(* CODESYS project Lift Structured Text New.project

Project tree, tasks and I/O mapping:
  CageTest : CODESYS Control Win V3, 3S - Smart Software Solutions GmbH, version 3.5.14.0
    application Application
      task CageTestTask (cyclic, interval t#20ms, priority 1) calls Simulatie, CageTestProgram
      visualisation Visualization
  DoorTest : CODESYS Control Win V3, 3S - Smart Software Solutions GmbH, version 3.5.14.0
    application Application
      libraries: Standard, * (System)
      task DoorTestTask (cyclic, interval t#20ms, priority 1) calls DoorTestProgram, Simulatie
      visualisation Visualization
  Elevator : CODESYS Control Win V3, 3S - Smart Software Solutions GmbH, version 3.5.14.0
    application Application
      libraries: Standard, * (System)
      task ElevatorTask (cyclic, interval t#20ms, priority 1) calls MainProgram, Simulatie
      visualisation Visualization
  Lift Besturing/
    program DoorTestProgram [ST]
    function block Door [ST]: goOpen, goClose, isClosed, cycle, initialaize, isOpen
    data type DoorStates
    program MainProgram [ST]
    function block Elevator [ST]: initialiaze, cycle
    data type CageStates
    function block Cage [ST]: initialaize, cycle, startTraveling, isUp, isDown, isTraveling
    program CageTestProgram [ST]
    data type ElevatorStates
  global variables GVL
  image pool ImagePool
  5ce3da45-db07-42e7-a21c-a00fff4ed8f6|C:\Users\Gerard\Desktop\MensenInLift.PNG
  5ce3da45-db07-42e7-a21c-a00fff4ed8f6|C:\Users\Gerard\Desktop\LiftDeur.PNG
  5ce3da45-db07-42e7-a21c-a00fff4ed8f6|C:\Users\Gerard\Desktop\Liftaandrijving.PNG
  5ce3da45-db07-42e7-a21c-a00fff4ed8f6|C:\Users\Gerard\Desktop\LiftDeurAandrijving.PNG
  Lift Simualtie/
    program Simulatie [ST]
  text list GlobalTextList
  visualisation Visualization
*)

// Lift Besturing/DoorStates
// Authour : G A Harkema
// Date:  february 15, 2017
// Version : 1.0
// States of the door
TYPE DoorStates :
(
	idle := 0,close, toOpen, open, toClose
);
END_TYPE

// Lift Besturing/CageStates
// Authour : G A Harkema
// Date:  february 15, 2017
// Version : 1.0
// States of the cage
TYPE CageStates :
(
	idle := 0, stationary, goUp, goDown  
);
END_TYPE

// Lift Besturing/ElevatorStates
// Authour : G A Harkema
// Date:  february 15, 2017
// Version : 1.0
// States of the cage
TYPE ElevatorStates :
(
	idle := 0, waitForChoise, closingDoor, traveling, openingDoor
);
END_TYPE

// GVL
VAR_GLOBAL
	Ix_BovenOproepKooi					: BOOL;
	Ix_BenedenOproepKooi				: BOOL;
	Ix_KooiGaNaarBoven					: BOOL;
	Ix_KooiGaNaarBeneden				: BOOL;
	Ix_KooiBoven						: BOOL;
	Ix_KooiBeneden						: BOOL;
	Qx_AandrijvingOmhoog				: BOOL;
	Qx_AandrijvingOmlaag				: BOOL;
	
	
	Ix_BenedenDeurOpen					: BOOL;
	Ix_BenedenDeurGesloten				: BOOL;
	Qx_BenedenDeurAandrijvingOpen		: BOOL;
	Qx_BenedenDeurAandrijvingSluiten	: BOOL;
	
	Ix_BovenDeurOpen					: BOOL;
	Ix_BovenDeurGesloten				: BOOL;
	Qx_BovenDeurAandrijvingOpen			: BOOL;
	Qx_BovenDeurAandrijvingSluiten		: BOOL;
	
	Ix_TestButton1						: BOOL;
	Ix_TestButton2						: BOOL;
	
	Qx_TestIndicator1					: BOOL;
	Qx_TestIndicator2					: BOOL;
	
END_VAR

// Lift Simualtie/Simulatie
// Programma		: Simulatie
// Project			: Lift
// Doel				: Simulatie functies voor de lift
// Auteur			: Gerard Harkema
// Versie			: 1.0
// Datum			: 15 oktober 2015

PROGRAM Simulatie
VAR

	Mw_PositieLiftInv					: INT := 0;
	Mw_PositieLift						: INT := 0;
	Mw_LiftBenedenCountValue			: INT := 250;

	Mw_BenedenPositieDeur				: INT := 0;
	Mw_BenedenPositieDeurCountValue		: INT := 100;

	Mw_BovenPositieDeur					: INT := 0;
	Mw_BovenPositieDeurCountValue		: INT := 100;

END_VAR


// Reizen lift omhoog
IF(GVL.Qx_AandrijvingOmhoog AND (NOT GVL.Ix_KooiBoven)) THEN
	Mw_PositieLiftInv := Mw_PositieLiftInv + 1;
END_IF

// Reizen lift omlaag
IF(GVL.Qx_AandrijvingOmlaag AND (NOT GVL.Ix_KooiBeneden)) THEN
	Mw_PositieLiftInv := Mw_PositieLiftInv - 1;
END_IF

Mw_PositieLift := Mw_LiftBenedenCountValue - Mw_PositieLiftInv;

// Detectie lift is boven
IF (Mw_PositieLiftInv >= Mw_LiftBenedenCountValue) THEN
	GVL.Ix_KooiBoven := TRUE;
ELSE
	GVL.Ix_KooiBoven := FALSE;	
END_IF
  

// Detectie lift is beneden
IF(Mw_PositieLiftInv <= 0) THEN
	GVL.Ix_KooiBeneden := TRUE;
ELSE
	GVL.Ix_KooiBeneden := FALSE;	
END_IF

// Inactief maken oproepknoppen
IF GVL.Ix_KooiBoven THEN
 Ix_BovenOproepKooi := FALSE;
 Ix_KooiGaNaarBoven := FALSE;
END_IF

IF GVL.Ix_KooiBeneden THEN
 Ix_BenedenOproepKooi := FALSE;
 Ix_KooiGaNaarBeneden := FALSE;
END_IF


//*********************************************
//                 Bovendeur
//*********************************************

// Bovendeur openen
IF(GVL.Qx_BovenDeurAandrijvingOpen AND (NOT GVL.Ix_BovenDeurOpen)) THEN
	Mw_BovenPositieDeur := Mw_BovenPositieDeur + 1;
END_IF

// Bovendeur sluiten
IF(GVL.Qx_BovenDeurAandrijvingSluiten AND (NOT GVL.Ix_BovenDeurGesloten)) THEN
	Mw_BovenPositieDeur := Mw_BovenPositieDeur - 1;
END_IF

IF (Mw_BovenPositieDeur >= Mw_BovenPositieDeurCountValue) THEN
	GVL.Ix_BovenDeurOpen := TRUE;
ELSE
	GVL.Ix_BovenDeurOpen := FALSE;	
END_IF
  

// Detectie bovendeur is gesloten
IF(Mw_BovenPositieDeur <= 0) THEN
	GVL.Ix_BovenDeurGesloten := TRUE;
ELSE
	GVL.Ix_BovenDeurGesloten := FALSE;	
END_IF

//*********************************************
//                 Benedendeur
//*********************************************

// Benedendeur openen
IF(GVL.Qx_BenedenDeurAandrijvingOpen AND (NOT GVL.Ix_BenedenDeurOpen)) THEN
	Mw_BenedenPositieDeur := Mw_BenedenPositieDeur + 1;
END_IF

// Benedendeur sluiten
IF(GVL.Qx_BenedenDeurAandrijvingSluiten AND (NOT GVL.Ix_BenedenDeurGesloten)) THEN
	Mw_BenedenPositieDeur := Mw_BenedenPositieDeur - 1;
END_IF

// Detectie Benedendeur is open
IF (Mw_BenedenPositieDeur >= Mw_BenedenPositieDeurCountValue) THEN
	GVL.Ix_BenedenDeurOpen := TRUE;
ELSE
	GVL.Ix_BenedenDeurOpen := FALSE;	
END_IF

// Detectie Benedendeur is gesloten
IF(Mw_BenedenPositieDeur <= 0) THEN
	GVL.Ix_BenedenDeurGesloten := TRUE;
ELSE
	GVL.Ix_BenedenDeurGesloten := FALSE;	
END_IF

END_PROGRAM

// Lift Besturing/CageTestProgram
// Authour : G A Harkema
// Date:  february 15, 2017
// Version : 1.0
// Testprogram for the cage

PROGRAM CageTestProgram
VAR
	theCage				: Cage;
	firstRun		 	: BOOL := TRUE;
END_VAR

IF firstRun THEN
	// make references to I/O
	theCage.initialaize();
	firstRun := FALSE;
END_IF

// Update inputs of the objects
theCage.xCageIsUp := gvl.Ix_KooiBoven;
theCage.xCageIsDown := gvl.Ix_KooiBeneden;

theCage.cycle();

// Update Outputs from the object
gvl.Qx_AandrijvingOmhoog := TheCage.xTransmissionUp;
gvl.Qx_AandrijvingOmlaag := TheCage.xTransmissionDown;

Qx_TestIndicator1 := theCage.isTraveling();

IF NOT theCage.isTraveling() THEN
	IF Ix_TestButton1 THEN // Handle button event
		Ix_TestButton1 := FALSE;
		theCage.startTraveling();
	END_IF
END_IF

END_PROGRAM

// Lift Besturing/Cage
// Authour : G A Harkema
// Date:  february 15, 2017
// Version : 1.0
// Class of the elevator

FUNCTION_BLOCK Cage
VAR
	eState								: CageStates := CageStates.idle;
END_VAR

VAR_INPUT
	xCageIsUp							: BOOL; 
	xCageIsDown							: BOOL; 
END_VAR

VAR_OUTPUT
	xTransmissionUp						: BOOL; 
	xTransmissionDown					: BOOL; 
END_VAR

// Statemachine of the cage
CASE eState OF

	CageStates.idle:
		xTransmissionDown := TRUE;  // powerup sequence
		eState := CageStates.goDown;


	CageStates.goDown:
		IF xCageIsDown THEN  // Handle downstair event
			xTransmissionDown := FALSE;
			eState := CageStates.stationary;
		END_IF
	
	CageStates.goUp:
		IF xCageIsUp THEN  // Handle upstairs event
			xTransmissionUp := FALSE;
			eState := CageStates.stationary;
		END_IF

	
END_CASE

// initialaize I/O
METHOD initialaize
VAR_INPUT
END_VAR
// Set default values
xTransmissionUp 	:= FALSE;
xTransmissionDown 	:= FALSE;
END_METHOD

// Update statemachine and I/O
METHOD cycle
VAR_INPUT
END_VAR
THIS^();
END_METHOD

// start traveling of cage
METHOD startTraveling
VAR_INPUT
END_VAR
IF eState = CageStates.stationary THEN
	
	// Check position of the cage and handle
	IF isUp() THEN
		xTransmissionDown := TRUE;
		eState := CageStates.goDown;
	END_IF
	
	IF isDown() THEN
		xTransmissionUp := TRUE;
		eState := CageStates.goUp;
	END_IF
	
END_IF
END_METHOD

// check upstairs methode
METHOD PUBLIC isUp : BOOL
VAR_INPUT
END_VAR
isUp := xCageIsUp;
END_METHOD

// check downstairs methode
METHOD PUBLIC isDown : BOOL
VAR_INPUT
END_VAR
isDown := xCageIsDown;
END_METHOD

// check traveling methode
METHOD PUBLIC isTraveling : BOOL
VAR_INPUT
END_VAR
isTraveling := NOT(eState = CageStates.stationary);
END_METHOD

END_FUNCTION_BLOCK

// Lift Besturing/Elevator
// Authour : G A Harkema
// Date:  february 15, 2017
// Version : 1.0
// Class of the elevator

FUNCTION_BLOCK Elevator
VAR_INPUT
	doorUpstairs   		: Door;
	doorDownstairs   	: Door;
	theCage				: Cage;
	initialiazed	 	: BOOL := FALSE;
	eState				: ElevatorStates := ElevatorStates.idle;
END_VAR

IF initialiazed THEN
	// Update statemachines and I/O
	doorUpstairs.cycle();
	doorDownstairs.cycle();
	theCage.cycle();
END_IF

METHOD initialiaze
VAR_INPUT
END_VAR
// make references to I/O
theCage.initialaize();
doorUpstairs.initialaize();
doorDownstairs.initialaize();

initialiazed := TRUE;
END_METHOD

// Update statemachine and I/O
METHOD cycle
VAR_INPUT
END_VAR
THIS^();

// Update inputs of the objects
theCage.xCageIsUp := gvl.Ix_KooiBoven;
theCage.xCageIsDown := gvl.Ix_KooiBeneden;

doorDownstairs.xDoorIsOpen := gvl.Ix_BenedenDeurOpen;
doorDownstairs.xDoorIsClose := gvl.Ix_BenedenDeurGesloten;

doorUpstairs.xDoorIsOpen := gvl.Ix_BovenDeurOpen;
doorUpstairs.xDoorIsClose := gvl.Ix_BovenDeurGesloten;

	
// Handle state machine
CASE eState OF
	ElevatorStates.idle:
		eState := ElevatorStates.waitForChoise;

	ElevatorStates.waitForChoise:
		IF theCage.isUp() THEN  // handle choise
			IF Ix_KooiGaNaarBeneden OR Ix_BenedenOproepKooi THEN
				doorUpstairs.goClose();
				eState := ElevatorStates.closingDoor;
			END_IF
		END_IF
		
		IF theCage.isDown() THEN
			IF Ix_KooiGaNaarBoven OR Ix_BovenOproepKooi THEN
				doorDownstairs.goClose();
				eState := ElevatorStates.closingDoor;
			END_IF
		END_IF

	ElevatorStates.closingDoor:
		IF doorUpstairs.isClosed() AND doorDownstairs.isClosed() THEN // handle doors closed
			theCage.startTraveling();
			eState := ElevatorStates.traveling;
		END_IF
	
	ElevatorStates.traveling:
		IF NOT theCage.isTraveling() THEN // handle arriving of cage
			IF theCage.isUp()  THEN
				doorUpstairs.goOpen();
				eState := ElevatorStates.openingDoor;
			END_IF
	
			IF theCage.isDown() THEN
				doorDownstairs.goOpen();
				eState := ElevatorStates.openingDoor;
			END_IF
		END_IF;

	ElevatorStates.openingDoor:
		IF doorUpstairs.isOpen() OR doorDownstairs.isOpen() THEN // Handle door open
			eState := ElevatorStates.waitForChoise;
		END_IF
END_CASE

// Update Outputs from the object
gvl.Qx_AandrijvingOmhoog := TheCage.xTransmissionUp;
gvl.Qx_AandrijvingOmlaag := TheCage.xTransmissionDown;

gvl.Qx_BenedenDeurAandrijvingOpen := doorDownstairs.xDoorOpening;
gvl.Qx_BenedenDeurAandrijvingSluiten := doorDownstairs.xDoorClosing;

gvl.Qx_BovenDeurAandrijvingOpen := doorUpstairs.xDoorOpening;
gvl.Qx_BovenDeurAandrijvingSluiten := doorUpstairs.xDoorClosing;
END_METHOD

END_FUNCTION_BLOCK

// Lift Besturing/Door
// Authour : G A Harkema
// Date:  february 15, 2017
// Version : 1.0
// Class of the door

FUNCTION_BLOCK Door
VAR
	eState							: DoorStates := DoorStates.idle;
END_VAR

VAR_INPUT
	xDoorIsOpen						: BOOL; 
	xDoorIsClose					: BOOL; 
END_VAR

VAR_OUTPUT
	xDoorOpening					: BOOL; 
	xDoorClosing					: BOOL; 
END_VAR

// Statemachine of the door
CASE eState OF
	DoorStates.toOpen :
		IF xDoorIsOpen THEN  // handle open event
			xDoorOpening := FALSE;
			eState := DoorStates.open;
		END_IF
	
	DoorStates.toClose :
		IF xDoorIsClose THEN // handle close event
			xDoorClosing := FALSE;
			eState := DoorStates.close;
		END_IF
	
END_CASE

// start door open action methode
METHOD PUBLIC goOpen
VAR_INPUT
END_VAR
// Trigger door
IF eState = DoorStates.close THEN
	eState := DoorStates.toOpen;  // Hnadle event
	xDoorOpening := TRUE;
END_IF
END_METHOD

// start close door action method
METHOD PUBLIC goClose
VAR_INPUT
END_VAR
// Trigger door when open
IF eState = DoorStates.open THEN
	eState := DoorStates.toClose;  // Handle event
	xDoorClosing := TRUE;
END_IF


// Trigger door when close
IF eState = DoorStates.idle THEN
	eState := DoorStates.toClose; // Hnadle event
	xDoorClosing := TRUE;
END_IF
END_METHOD

// check door closed method
METHOD PUBLIC isClosed : BOOL
VAR_INPUT
END_VAR
isClosed := eState = DoorStates.close;
END_METHOD

// Update statemachine and I/O
METHOD cycle
VAR_INPUT
END_VAR
THIS^();
END_METHOD

// initialaize I/O
METHOD initialaize
VAR_INPUT
END_VAR

xDoorOpening := FALSE;
xDoorClosing := FALSE;
	

// Close the door	
goClose();
END_METHOD

// check door opened method
METHOD isOpen : BOOL
VAR_INPUT
END_VAR
isOpen := eState = DoorStates.open;
END_METHOD

END_FUNCTION_BLOCK

// Lift Besturing/DoorTestProgram
// Authour : G A Harkema
// Date:  february 15, 2017
// Version : 1.0
// Testprogram for the doors

PROGRAM DoorTestProgram
VAR
	doorUpstairs   		: Door;
	doorDownstairs   	: Door;
	firstRun		 	: BOOL := TRUE;
END_VAR

IF firstRun THEN
	// make references to I/O
	doorUpstairs.initialaize();
	doorDownstairs.initialaize();
	firstRun := FALSE;
END_IF

// Update inputs of the objects
doorDownstairs.xDoorIsOpen := gvl.Ix_BenedenDeurOpen;
doorDownstairs.xDoorIsClose := gvl.Ix_BenedenDeurGesloten;

doorUpstairs.xDoorIsOpen := gvl.Ix_BovenDeurOpen;
doorUpstairs.xDoorIsClose := gvl.Ix_BovenDeurGesloten;

// update I/O
doorUpstairs.cycle();
doorDownstairs.cycle();

// Update Outputs from the object
gvl.Qx_BenedenDeurAandrijvingOpen := doorDownstairs.xDoorOpening;
gvl.Qx_BenedenDeurAandrijvingSluiten := doorDownstairs.xDoorClosing;

gvl.Qx_BovenDeurAandrijvingOpen := doorUpstairs.xDoorOpening;
gvl.Qx_BovenDeurAandrijvingSluiten := doorUpstairs.xDoorClosing;

IF Ix_TestButton1 THEN
	Ix_TestButton1 := FALSE; // Handle button event
	doorUpstairs.goOpen();
	doorDownstairs.goClose();
END_IF

IF Ix_TestButton2 THEN
	Ix_TestButton2 := FALSE; // Handle button event
	doorUpstairs.goClose();
	doorDownstairs.goOpen();
END_IF

END_PROGRAM

// Lift Besturing/MainProgram
// Authour : G A Harkema
// Date:  february 15, 2017
// Version : 1.0
// Main program of the elevator

PROGRAM MainProgram
VAR
	// only one object is created in the main program
	theElevator			: Elevator;
	firstRun		 	: BOOL := TRUE;
END_VAR

IF firstRun THEN
	theElevator.initialiaze ();
	firstRun := FALSE;
END_IF


// update statemachines and I/O
theElevator.cycle();

END_PROGRAM

// CageTest/Application/Visualization
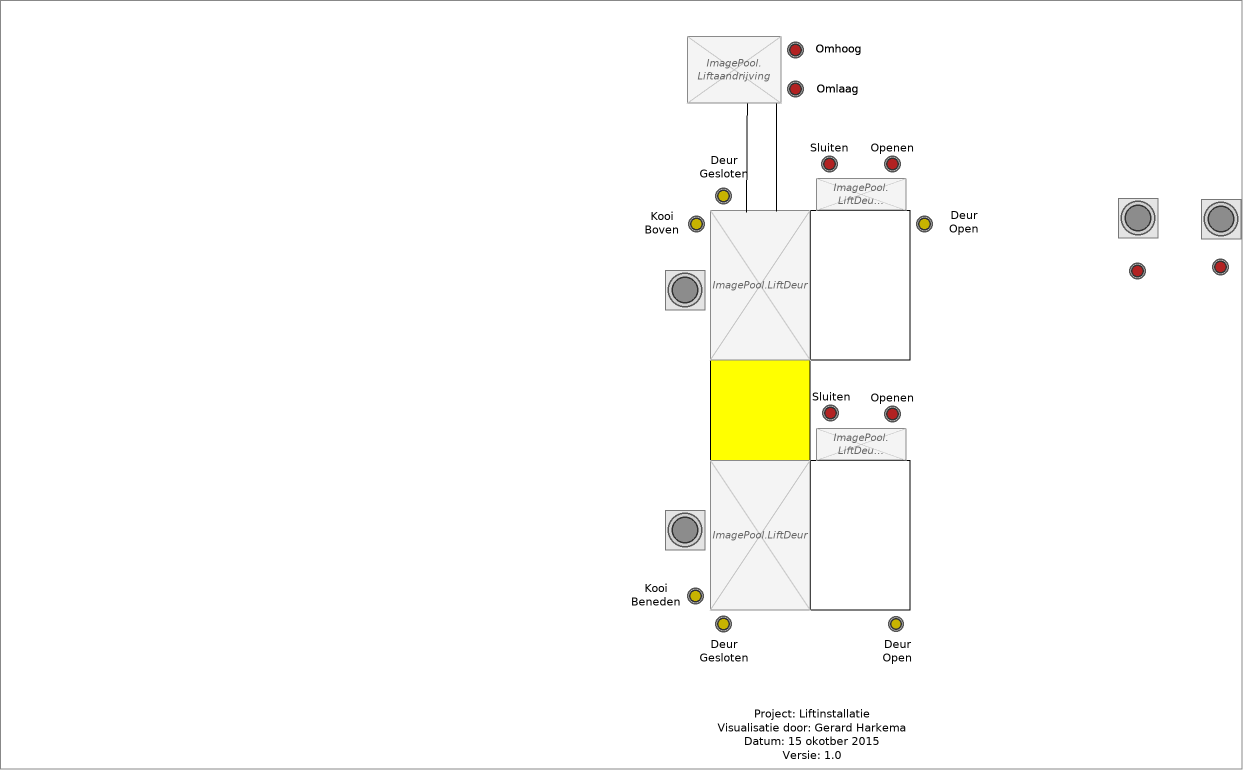
VISUALIZATION Visualization  // 1243x770
    Rectangle (810,460 100x150)
    Rectangle (810,210 100x150)
    Rectangle (710,210 100x400)
    PushSwitch (665,270 40x40), tooltip "Oproep Boven", variable: Ix_BovenOproepKooi, behaviour: TOGGLE, style: Switch-PushSwitch-Gray
    PushSwitch (665,510 40x40), tooltip "Oproep Beneden", variable: Ix_BenedenOproepKooi, behaviour: TOGGLE, style: Switch-PushSwitch-Gray
    Group (710,210 100x150)
        p2738717112: Simulatie.Mw_PositieLift
        Rectangle (0,0 100x150)
        Image (6,0 89x150), image: ImagePool.MensenInLift
        PushSwitch (5,100 30x30), tooltip "Ga naar beneden", variable: Ix_KooiGaNaarBeneden, behaviour: TOGGLE, style: Switch-PushSwitch-Gray
        PushSwitch (5,60 30x30), tooltip "Ga naar Boven", variable: Ix_KooiGaNaarBoven, behaviour: TOGGLE, style: Switch-PushSwitch-Gray
    Rectangle (710,210 100x150)
    Image (716,210 89x150), image: ImagePool.MensenInLift
    PushSwitch (715,310 30x30), tooltip "Ga naar beneden", variable: Ix_KooiGaNaarBeneden, behaviour: TOGGLE, style: Switch-PushSwitch-Gray
    PushSwitch (715,270 30x30), tooltip "Ga naar Boven", variable: Ix_KooiGaNaarBoven, behaviour: TOGGLE, style: Switch-PushSwitch-Gray
    Lamp1 (714,186 19x20), variable: Ix_BovenDeurGesloten, style: Lamp-Lamp1-Yellow
    Lamp1 (915,214 19x20), variable: Ix_BovenDeurOpen, style: Lamp-Lamp1-Yellow
    Lamp1 (687,214 19x20), variable: Ix_KooiBoven, style: Lamp-Lamp1-Yellow
    Lamp1 (686,586 19x20), variable: Ix_KooiBeneden, style: Lamp-Lamp1-Yellow
    Lamp1 (714,614 19x20), variable: Ix_BenedenDeurGesloten, style: Lamp-Lamp1-Yellow
    Lamp1 (887,614 18x20), variable: Ix_BenedenDeurOpen, style: Lamp-Lamp1-Yellow
    Label (682,152 84x30), "Deur Gesloten"
    Label (937,207 54x30), "Deur Open"
    Label (640,208 44x30), "Kooi Boven"
    Label (629,580 54x30), "Kooi Beneden"
    Label (693,636 62x30), "Deur Gesloten"
    Label (875,636 45x30), "Deur Open"
    Group (710,210 100x150)
        p3560616238: Simulatie.Mw_BovenPositieDeur
        Rectangle (0,0 100x150)
        Image (0,0 100x150), image: ImagePool.LiftDeur
    Group (710,460 100x150)
        p3560616238: Simulatie.Mw_BenedenPositieDeur
        Rectangle (0,0 100x150)
        Image (0,0 100x150), image: ImagePool.LiftDeur
    Line (747,83) (746,212)
    Line (776,82) (776,211)
    Group (687,34 182x70)
        Image (0,2 94x67), image: ImagePool.Liftaandrijving
        Lamp1 (99,6 19x20), variable: Qx_AandrijvingOmhoog, style: Lamp-Lamp1-Red
        Lamp1 (99,45 19x20), variable: Qx_AandrijvingOmlaag, style: Lamp-Lamp1-Red
        Label (121,0 61x30), "Omhoog"
        Label (123,40 55x30), "Omlaag"
    Image (687,36 94x67), image: ImagePool.Liftaandrijving
    Lamp1 (786,40 19x20), variable: Qx_AandrijvingOmhoog, style: Lamp-Lamp1-Red
    Lamp1 (786,79 19x20), variable: Qx_AandrijvingOmlaag, style: Lamp-Lamp1-Red
    Label (808,34 61x30), "Omhoog"
    Label (810,74 55x30), "Omlaag"
    Group (816,154 90x56)
        Image (0,24 90x32), image: ImagePool.LiftDeurAandrijving
        Lamp1 (4,0 19x20), variable: Qx_BovenDeurAandrijvingSluiten, style: Lamp-Lamp1-Red
        Lamp1 (67,0 19x20), variable: Qx_BovenDeurAandrijvingOpen, style: Lamp-Lamp1-Red
    Image (816,178 90x32), image: ImagePool.LiftDeurAandrijving
    Lamp1 (820,154 19x20), variable: Qx_BovenDeurAandrijvingSluiten, style: Lamp-Lamp1-Red
    Lamp1 (883,154 19x20), variable: Qx_BovenDeurAandrijvingOpen, style: Lamp-Lamp1-Red
    Group (816,403 90x57)
        Image (0,25 90x32), image: ImagePool.LiftDeurAandrijving
        Lamp1 (5,0 19x20), variable: Qx_BenedenDeurAandrijvingSluiten, style: Lamp-Lamp1-Red
        Lamp1 (67,1 19x20), variable: Qx_BenedenDeurAandrijvingOpen, style: Lamp-Lamp1-Red
    Image (816,428 90x32), image: ImagePool.LiftDeurAandrijving
    Lamp1 (821,403 19x20), variable: Qx_BenedenDeurAandrijvingSluiten, style: Lamp-Lamp1-Red
    Lamp1 (883,404 19x20), variable: Qx_BenedenDeurAandrijvingOpen, style: Lamp-Lamp1-Red
    Label (812,382 39x30), "Sluiten"
    Label (810,133 39x30), "Sluiten"
    Label (867,383 51x30), "Openen"
    Label (867,133 51x30), "Openen"
    Label (712,701 200x67), "Project: Liftinstallatie Visualisatie door: Gerard Harkema Datum: 15 okotber 2015 Versie: 1.0"
    PushSwitch (1118,198 40x40), tooltip "Test Button 1", variable: Ix_TestButton1, behaviour: TOGGLE, style: Switch-PushSwitch-Gray
    PushSwitch (1201,199 40x40), tooltip "Test Button 2", variable: Ix_TestButton2, behaviour: TOGGLE, style: Switch-PushSwitch-Gray
    Lamp1 (1128,261 19x20), variable: Qx_TestIndicator1, style: Lamp-Lamp1-Red
    Lamp1 (1211,257 19x20), variable: Qx_TestIndicator2, style: Lamp-Lamp1-Red
END_VISUALIZATION

// DoorTest/Application/Visualization
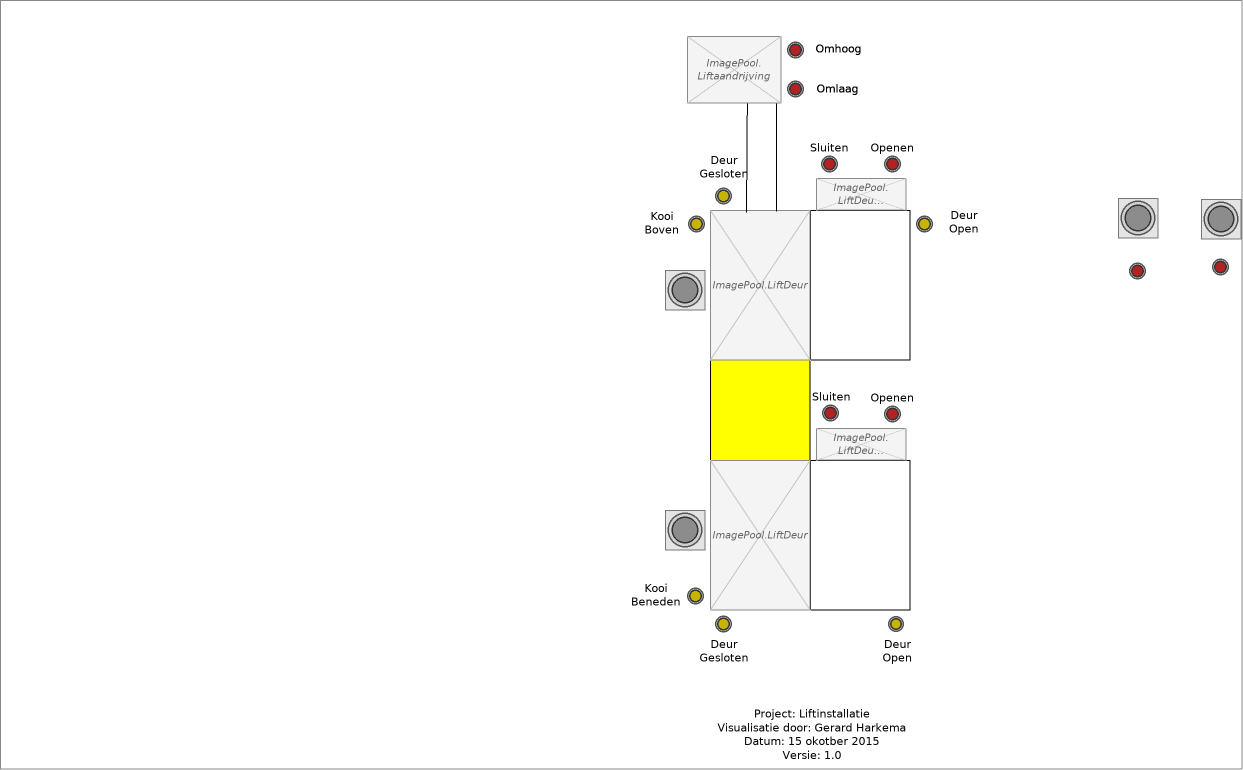
VISUALIZATION Visualization  // 1243x770
    Rectangle (810,460 100x150)
    Rectangle (810,210 100x150)
    Rectangle (710,210 100x400)
    PushSwitch (665,270 40x40), tooltip "Oproep Boven", variable: Ix_BovenOproepKooi, behaviour: TOGGLE, style: Switch-PushSwitch-Gray
    PushSwitch (665,510 40x40), tooltip "Oproep Beneden", variable: Ix_BenedenOproepKooi, behaviour: TOGGLE, style: Switch-PushSwitch-Gray
    Group (710,210 100x150)
        p2738717112: Simulatie.Mw_PositieLift
        Rectangle (0,0 100x150)
        Image (6,0 89x150), image: ImagePool.MensenInLift
        PushSwitch (5,100 30x30), tooltip "Ga naar beneden", variable: Ix_KooiGaNaarBeneden, behaviour: TOGGLE, style: Switch-PushSwitch-Gray
        PushSwitch (5,60 30x30), tooltip "Ga naar Boven", variable: Ix_KooiGaNaarBoven, behaviour: TOGGLE, style: Switch-PushSwitch-Gray
    Rectangle (710,210 100x150)
    Image (716,210 89x150), image: ImagePool.MensenInLift
    PushSwitch (715,310 30x30), tooltip "Ga naar beneden", variable: Ix_KooiGaNaarBeneden, behaviour: TOGGLE, style: Switch-PushSwitch-Gray
    PushSwitch (715,270 30x30), tooltip "Ga naar Boven", variable: Ix_KooiGaNaarBoven, behaviour: TOGGLE, style: Switch-PushSwitch-Gray
    Lamp1 (714,186 19x20), variable: Ix_BovenDeurGesloten, style: Lamp-Lamp1-Yellow
    Lamp1 (915,214 19x20), variable: Ix_BovenDeurOpen, style: Lamp-Lamp1-Yellow
    Lamp1 (687,214 19x20), variable: Ix_KooiBoven, style: Lamp-Lamp1-Yellow
    Lamp1 (686,586 19x20), variable: Ix_KooiBeneden, style: Lamp-Lamp1-Yellow
    Lamp1 (714,614 19x20), variable: Ix_BenedenDeurGesloten, style: Lamp-Lamp1-Yellow
    Lamp1 (887,614 18x20), variable: Ix_BenedenDeurOpen, style: Lamp-Lamp1-Yellow
    Label (682,152 84x30), "Deur Gesloten"
    Label (937,207 54x30), "Deur Open"
    Label (640,208 44x30), "Kooi Boven"
    Label (629,580 54x30), "Kooi Beneden"
    Label (693,636 62x30), "Deur Gesloten"
    Label (875,636 45x30), "Deur Open"
    Group (710,210 100x150)
        p3560616238: Simulatie.Mw_BovenPositieDeur
        Rectangle (0,0 100x150)
        Image (0,0 100x150), image: ImagePool.LiftDeur
    Group (710,460 100x150)
        p3560616238: Simulatie.Mw_BenedenPositieDeur
        Rectangle (0,0 100x150)
        Image (0,0 100x150), image: ImagePool.LiftDeur
    Line (747,83) (746,212)
    Line (776,82) (776,211)
    Group (687,34 182x70)
        Image (0,2 94x67), image: ImagePool.Liftaandrijving
        Lamp1 (99,6 19x20), variable: Qx_AandrijvingOmhoog, style: Lamp-Lamp1-Red
        Lamp1 (99,45 19x20), variable: Qx_AandrijvingOmlaag, style: Lamp-Lamp1-Red
        Label (121,0 61x30), "Omhoog"
        Label (123,40 55x30), "Omlaag"
    Image (687,36 94x67), image: ImagePool.Liftaandrijving
    Lamp1 (786,40 19x20), variable: Qx_AandrijvingOmhoog, style: Lamp-Lamp1-Red
    Lamp1 (786,79 19x20), variable: Qx_AandrijvingOmlaag, style: Lamp-Lamp1-Red
    Label (808,34 61x30), "Omhoog"
    Label (810,74 55x30), "Omlaag"
    Group (816,154 90x56)
        Image (0,24 90x32), image: ImagePool.LiftDeurAandrijving
        Lamp1 (4,0 19x20), variable: Qx_BovenDeurAandrijvingSluiten, style: Lamp-Lamp1-Red
        Lamp1 (67,0 19x20), variable: Qx_BovenDeurAandrijvingOpen, style: Lamp-Lamp1-Red
    Image (816,178 90x32), image: ImagePool.LiftDeurAandrijving
    Lamp1 (820,154 19x20), variable: Qx_BovenDeurAandrijvingSluiten, style: Lamp-Lamp1-Red
    Lamp1 (883,154 19x20), variable: Qx_BovenDeurAandrijvingOpen, style: Lamp-Lamp1-Red
    Group (816,403 90x57)
        Image (0,25 90x32), image: ImagePool.LiftDeurAandrijving
        Lamp1 (5,0 19x20), variable: Qx_BenedenDeurAandrijvingSluiten, style: Lamp-Lamp1-Red
        Lamp1 (67,1 19x20), variable: Qx_BenedenDeurAandrijvingOpen, style: Lamp-Lamp1-Red
    Image (816,428 90x32), image: ImagePool.LiftDeurAandrijving
    Lamp1 (821,403 19x20), variable: Qx_BenedenDeurAandrijvingSluiten, style: Lamp-Lamp1-Red
    Lamp1 (883,404 19x20), variable: Qx_BenedenDeurAandrijvingOpen, style: Lamp-Lamp1-Red
    Label (812,382 39x30), "Sluiten"
    Label (810,133 39x30), "Sluiten"
    Label (867,383 51x30), "Openen"
    Label (867,133 51x30), "Openen"
    Label (712,701 200x67), "Project: Liftinstallatie Visualisatie door: Gerard Harkema Datum: 15 okotber 2015 Versie: 1.0"
    PushSwitch (1118,198 40x40), tooltip "Test Button 1", variable: Ix_TestButton1, behaviour: TOGGLE, style: Switch-PushSwitch-Gray
    PushSwitch (1201,199 40x40), tooltip "Test Button 2", variable: Ix_TestButton2, behaviour: TOGGLE, style: Switch-PushSwitch-Gray
    Lamp1 (1128,261 19x20), variable: Qx_TestIndicator1, style: Lamp-Lamp1-Red
    Lamp1 (1211,257 19x20), variable: Qx_TestIndicator2, style: Lamp-Lamp1-Red
END_VISUALIZATION

// /Visualization
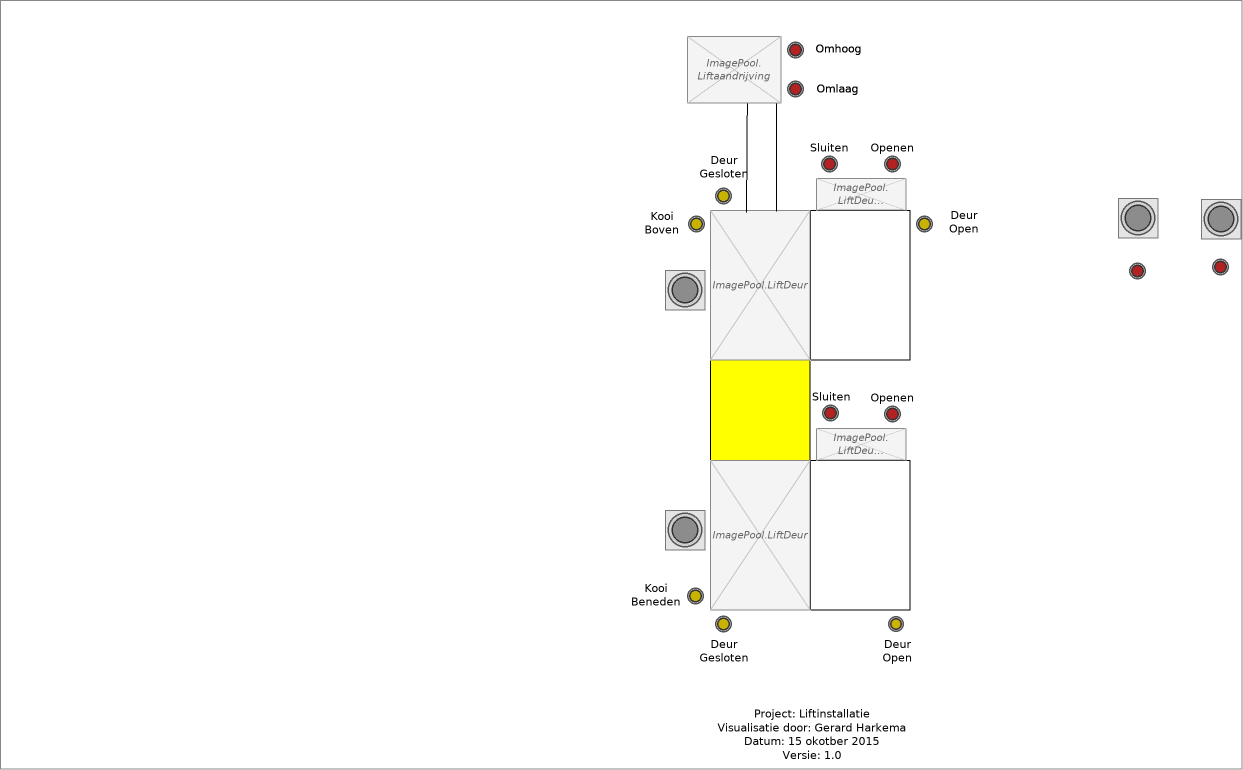
VISUALIZATION Visualization  // 1243x770
    Rectangle (810,460 100x150)
    Rectangle (810,210 100x150)
    Rectangle (710,210 100x400)
    PushSwitch (665,270 40x40), tooltip "Oproep Boven", variable: Ix_BovenOproepKooi, behaviour: TOGGLE, style: Switch-PushSwitch-Gray
    PushSwitch (665,510 40x40), tooltip "Oproep Beneden", variable: Ix_BenedenOproepKooi, behaviour: TOGGLE, style: Switch-PushSwitch-Gray
    Group (710,210 100x150)
        p2738717112: Simulatie.Mw_PositieLift
        Rectangle (0,0 100x150)
        Image (6,0 89x150), image: ImagePool.MensenInLift
        PushSwitch (5,100 30x30), tooltip "Ga naar beneden", variable: Ix_KooiGaNaarBeneden, behaviour: TOGGLE, style: Switch-PushSwitch-Gray
        PushSwitch (5,60 30x30), tooltip "Ga naar Boven", variable: Ix_KooiGaNaarBoven, behaviour: TOGGLE, style: Switch-PushSwitch-Gray
    Rectangle (710,210 100x150)
    Image (716,210 89x150), image: ImagePool.MensenInLift
    PushSwitch (715,310 30x30), tooltip "Ga naar beneden", variable: Ix_KooiGaNaarBeneden, behaviour: TOGGLE, style: Switch-PushSwitch-Gray
    PushSwitch (715,270 30x30), tooltip "Ga naar Boven", variable: Ix_KooiGaNaarBoven, behaviour: TOGGLE, style: Switch-PushSwitch-Gray
    Lamp1 (714,186 19x20), variable: Ix_BovenDeurGesloten, style: Lamp-Lamp1-Yellow
    Lamp1 (915,214 19x20), variable: Ix_BovenDeurOpen, style: Lamp-Lamp1-Yellow
    Lamp1 (687,214 19x20), variable: Ix_KooiBoven, style: Lamp-Lamp1-Yellow
    Lamp1 (686,586 19x20), variable: Ix_KooiBeneden, style: Lamp-Lamp1-Yellow
    Lamp1 (714,614 19x20), variable: Ix_BenedenDeurGesloten, style: Lamp-Lamp1-Yellow
    Lamp1 (887,614 18x20), variable: Ix_BenedenDeurOpen, style: Lamp-Lamp1-Yellow
    Label (682,152 84x30), "Deur Gesloten"
    Label (937,207 54x30), "Deur Open"
    Label (640,208 44x30), "Kooi Boven"
    Label (629,580 54x30), "Kooi Beneden"
    Label (693,636 62x30), "Deur Gesloten"
    Label (875,636 45x30), "Deur Open"
    Group (710,210 100x150)
        p3560616238: Simulatie.Mw_BovenPositieDeur
        Rectangle (0,0 100x150)
        Image (0,0 100x150), image: ImagePool.LiftDeur
    Group (710,460 100x150)
        p3560616238: Simulatie.Mw_BenedenPositieDeur
        Rectangle (0,0 100x150)
        Image (0,0 100x150), image: ImagePool.LiftDeur
    Line (747,83) (746,212)
    Line (776,82) (776,211)
    Group (687,34 182x70)
        Image (0,2 94x67), image: ImagePool.Liftaandrijving
        Lamp1 (99,6 19x20), variable: Qx_AandrijvingOmhoog, style: Lamp-Lamp1-Red
        Lamp1 (99,45 19x20), variable: Qx_AandrijvingOmlaag, style: Lamp-Lamp1-Red
        Label (121,0 61x30), "Omhoog"
        Label (123,40 55x30), "Omlaag"
    Image (687,36 94x67), image: ImagePool.Liftaandrijving
    Lamp1 (786,40 19x20), variable: Qx_AandrijvingOmhoog, style: Lamp-Lamp1-Red
    Lamp1 (786,79 19x20), variable: Qx_AandrijvingOmlaag, style: Lamp-Lamp1-Red
    Label (808,34 61x30), "Omhoog"
    Label (810,74 55x30), "Omlaag"
    Group (816,154 90x56)
        Image (0,24 90x32), image: ImagePool.LiftDeurAandrijving
        Lamp1 (4,0 19x20), variable: Qx_BovenDeurAandrijvingSluiten, style: Lamp-Lamp1-Red
        Lamp1 (67,0 19x20), variable: Qx_BovenDeurAandrijvingOpen, style: Lamp-Lamp1-Red
    Image (816,178 90x32), image: ImagePool.LiftDeurAandrijving
    Lamp1 (820,154 19x20), variable: Qx_BovenDeurAandrijvingSluiten, style: Lamp-Lamp1-Red
    Lamp1 (883,154 19x20), variable: Qx_BovenDeurAandrijvingOpen, style: Lamp-Lamp1-Red
    Group (816,403 90x57)
        Image (0,25 90x32), image: ImagePool.LiftDeurAandrijving
        Lamp1 (5,0 19x20), variable: Qx_BenedenDeurAandrijvingSluiten, style: Lamp-Lamp1-Red
        Lamp1 (67,1 19x20), variable: Qx_BenedenDeurAandrijvingOpen, style: Lamp-Lamp1-Red
    Image (816,428 90x32), image: ImagePool.LiftDeurAandrijving
    Lamp1 (821,403 19x20), variable: Qx_BenedenDeurAandrijvingSluiten, style: Lamp-Lamp1-Red
    Lamp1 (883,404 19x20), variable: Qx_BenedenDeurAandrijvingOpen, style: Lamp-Lamp1-Red
    Label (812,382 39x30), "Sluiten"
    Label (810,133 39x30), "Sluiten"
    Label (867,383 51x30), "Openen"
    Label (867,133 51x30), "Openen"
    Label (712,701 200x67), "Project: Liftinstallatie Visualisatie door: Gerard Harkema Datum: 15 okotber 2015 Versie: 1.0"
    PushSwitch (1118,198 40x40), tooltip "Test Button 1", variable: Ix_TestButton1, behaviour: TOGGLE, style: Switch-PushSwitch-Gray
    PushSwitch (1201,199 40x40), tooltip "Test Button 2", variable: Ix_TestButton2, behaviour: TOGGLE, style: Switch-PushSwitch-Gray
    Lamp1 (1128,261 19x20), variable: Qx_TestIndicator1, style: Lamp-Lamp1-Red
    Lamp1 (1211,257 19x20), variable: Qx_TestIndicator2, style: Lamp-Lamp1-Red
END_VISUALIZATION

// Elevator/Application/Visualization
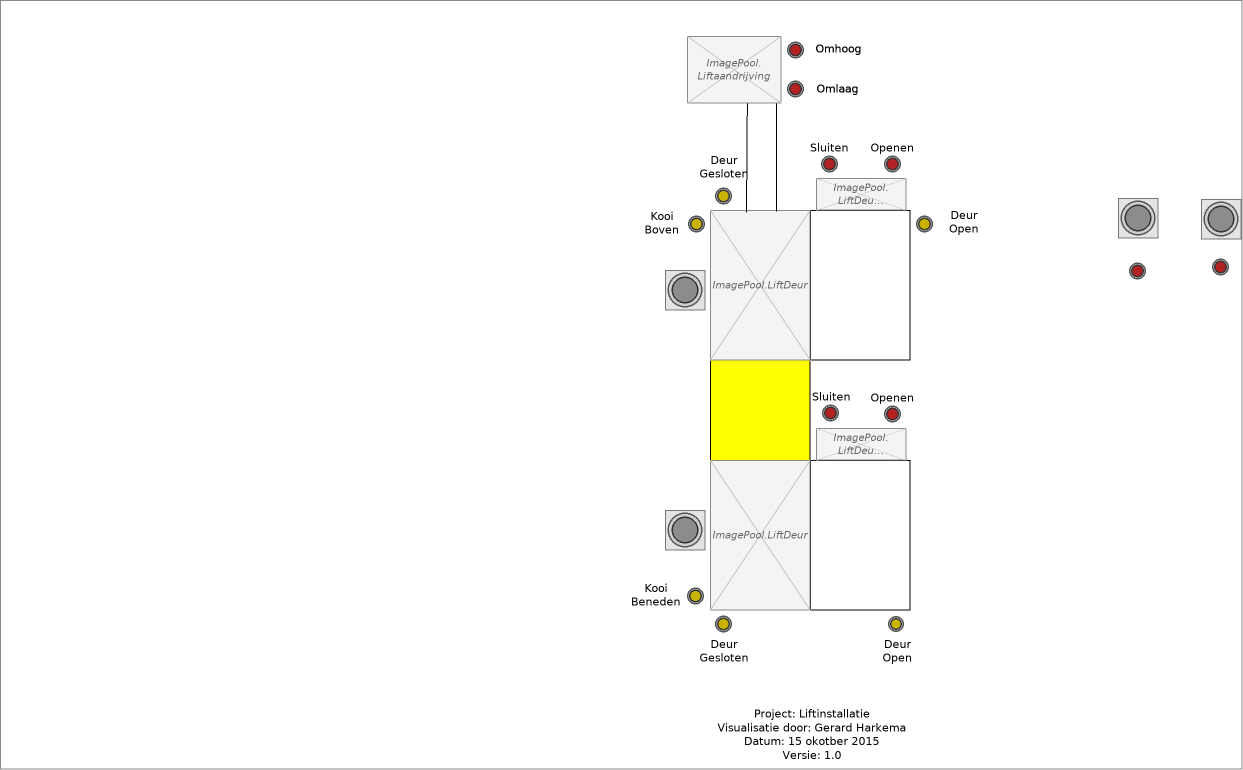
VISUALIZATION Visualization  // 1243x770
    Rectangle (810,460 100x150)
    Rectangle (810,210 100x150)
    Rectangle (710,210 100x400)
    PushSwitch (665,270 40x40), tooltip "Oproep Boven", variable: Ix_BovenOproepKooi, behaviour: TOGGLE, style: Switch-PushSwitch-Gray
    PushSwitch (665,510 40x40), tooltip "Oproep Beneden", variable: Ix_BenedenOproepKooi, behaviour: TOGGLE, style: Switch-PushSwitch-Gray
    Group (710,210 100x150)
        p2738717112: Simulatie.Mw_PositieLift
        Rectangle (0,0 100x150)
        Image (6,0 89x150), image: ImagePool.MensenInLift
        PushSwitch (5,100 30x30), tooltip "Ga naar beneden", variable: Ix_KooiGaNaarBeneden, behaviour: TOGGLE, style: Switch-PushSwitch-Gray
        PushSwitch (5,60 30x30), tooltip "Ga naar Boven", variable: Ix_KooiGaNaarBoven, behaviour: TOGGLE, style: Switch-PushSwitch-Gray
    Rectangle (710,210 100x150)
    Image (716,210 89x150), image: ImagePool.MensenInLift
    PushSwitch (715,310 30x30), tooltip "Ga naar beneden", variable: Ix_KooiGaNaarBeneden, behaviour: TOGGLE, style: Switch-PushSwitch-Gray
    PushSwitch (715,270 30x30), tooltip "Ga naar Boven", variable: Ix_KooiGaNaarBoven, behaviour: TOGGLE, style: Switch-PushSwitch-Gray
    Lamp1 (714,186 19x20), variable: Ix_BovenDeurGesloten, style: Lamp-Lamp1-Yellow
    Lamp1 (915,214 19x20), variable: Ix_BovenDeurOpen, style: Lamp-Lamp1-Yellow
    Lamp1 (687,214 19x20), variable: Ix_KooiBoven, style: Lamp-Lamp1-Yellow
    Lamp1 (686,586 19x20), variable: Ix_KooiBeneden, style: Lamp-Lamp1-Yellow
    Lamp1 (714,614 19x20), variable: Ix_BenedenDeurGesloten, style: Lamp-Lamp1-Yellow
    Lamp1 (887,614 18x20), variable: Ix_BenedenDeurOpen, style: Lamp-Lamp1-Yellow
    Label (682,152 84x30), "Deur Gesloten"
    Label (937,207 54x30), "Deur Open"
    Label (640,208 44x30), "Kooi Boven"
    Label (629,580 54x30), "Kooi Beneden"
    Label (693,636 62x30), "Deur Gesloten"
    Label (875,636 45x30), "Deur Open"
    Group (710,210 100x150)
        p3560616238: Simulatie.Mw_BovenPositieDeur
        Rectangle (0,0 100x150)
        Image (0,0 100x150), image: ImagePool.LiftDeur
    Group (710,460 100x150)
        p3560616238: Simulatie.Mw_BenedenPositieDeur
        Rectangle (0,0 100x150)
        Image (0,0 100x150), image: ImagePool.LiftDeur
    Line (747,83) (746,212)
    Line (776,82) (776,211)
    Group (687,34 182x70)
        Image (0,2 94x67), image: ImagePool.Liftaandrijving
        Lamp1 (99,6 19x20), variable: Qx_AandrijvingOmhoog, style: Lamp-Lamp1-Red
        Lamp1 (99,45 19x20), variable: Qx_AandrijvingOmlaag, style: Lamp-Lamp1-Red
        Label (121,0 61x30), "Omhoog"
        Label (123,40 55x30), "Omlaag"
    Image (687,36 94x67), image: ImagePool.Liftaandrijving
    Lamp1 (786,40 19x20), variable: Qx_AandrijvingOmhoog, style: Lamp-Lamp1-Red
    Lamp1 (786,79 19x20), variable: Qx_AandrijvingOmlaag, style: Lamp-Lamp1-Red
    Label (808,34 61x30), "Omhoog"
    Label (810,74 55x30), "Omlaag"
    Group (816,154 90x56)
        Image (0,24 90x32), image: ImagePool.LiftDeurAandrijving
        Lamp1 (4,0 19x20), variable: Qx_BovenDeurAandrijvingSluiten, style: Lamp-Lamp1-Red
        Lamp1 (67,0 19x20), variable: Qx_BovenDeurAandrijvingOpen, style: Lamp-Lamp1-Red
    Image (816,178 90x32), image: ImagePool.LiftDeurAandrijving
    Lamp1 (820,154 19x20), variable: Qx_BovenDeurAandrijvingSluiten, style: Lamp-Lamp1-Red
    Lamp1 (883,154 19x20), variable: Qx_BovenDeurAandrijvingOpen, style: Lamp-Lamp1-Red
    Group (816,403 90x57)
        Image (0,25 90x32), image: ImagePool.LiftDeurAandrijving
        Lamp1 (5,0 19x20), variable: Qx_BenedenDeurAandrijvingSluiten, style: Lamp-Lamp1-Red
        Lamp1 (67,1 19x20), variable: Qx_BenedenDeurAandrijvingOpen, style: Lamp-Lamp1-Red
    Image (816,428 90x32), image: ImagePool.LiftDeurAandrijving
    Lamp1 (821,403 19x20), variable: Qx_BenedenDeurAandrijvingSluiten, style: Lamp-Lamp1-Red
    Lamp1 (883,404 19x20), variable: Qx_BenedenDeurAandrijvingOpen, style: Lamp-Lamp1-Red
    Label (812,382 39x30), "Sluiten"
    Label (810,133 39x30), "Sluiten"
    Label (867,383 51x30), "Openen"
    Label (867,133 51x30), "Openen"
    Label (712,701 200x67), "Project: Liftinstallatie Visualisatie door: Gerard Harkema Datum: 15 okotber 2015 Versie: 1.0"
    PushSwitch (1118,198 40x40), tooltip "Test Button 1", variable: Ix_TestButton1, behaviour: TOGGLE, style: Switch-PushSwitch-Gray
    PushSwitch (1201,199 40x40), tooltip "Test Button 2", variable: Ix_TestButton2, behaviour: TOGGLE, style: Switch-PushSwitch-Gray
    Lamp1 (1128,261 19x20), variable: Qx_TestIndicator1, style: Lamp-Lamp1-Red
    Lamp1 (1211,257 19x20), variable: Qx_TestIndicator2, style: Lamp-Lamp1-Red
END_VISUALIZATION
